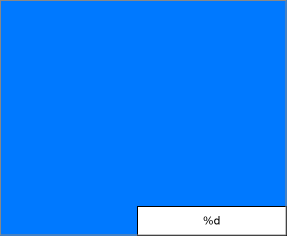
VISUALIZATION Main_Visu  // 287x236
    Rectangle (137,206 150x30), "%d", text variable: MAIN.iTest
END_VISUALIZATION

(* stored: Version 1.1.0.1, ProductVersion 3.1.4024.12
   Visu Main_Visu: Id {c6073acc-8d8b-4725-badf-f1a04931f1dd} *)
